(* PLC project passing_sensor, Dassault Systèmes ControlBuild 2024x *)
(* stored: creationDateTime 2023-10-03T11:13:57-01:00 *)

FUNCTION_BLOCK tri_chain.passing_sensor
  VAR_INPUT
    sensorSupply : BOOL := true;
  END_VAR
  VAR_OUTPUT
    passing : BOOL := false;
  END_VAR
  VAR
    status_act_prod : DINT := 0;
    m11 : REAL := 1.0;
    m12 : REAL := 0.0;
    m13 : REAL := 0.0;
    m14 : REAL := 0.0;
    m21 : REAL := 0.0;
    m22 : REAL := 1.0;
    m23 : REAL := 0.0;
    m24 : REAL := 0.0;
    m31 : REAL := 0.0;
    m32 : REAL := 0.0;
    m33 : REAL := 1.0;
    m34 : REAL := 0.0;
    m41 : REAL := 0.0;
    m42 : REAL := 0.0;
    m43 : REAL := 0.0;
    m44 : REAL := 1.0;
    px : REAL := 0.0;
    py : REAL := 0.0;
    pz : REAL := 0.0;
    dx : REAL := 0.0;
    dy : REAL := 0.0;
    dz : REAL := 0.0;
    detection : BOOL := false;
  END_VAR
  VAR CONSTANT
    passingLogic : BOOL := true;
  END_VAR
  VAR
    d_passing : BOOL := false;
    v_d_passing : BOOL := true;
  END_VAR


ACTION C_source_code:
/* ----------------------------------------------------------------	*/
/* Type : Model of Operative Behaviour					*/
/* Category :  Sensors							*/
/* Author : Dassault Systemes						*/
/* Update date : June 2018							*/
/* ----------------------------------------------------------------	*/
/* This module simulates the bahaviour of a  passing sensor 		*/
/*	for products.								*/
/* This module is an "actor".						*/
/* If it interacts with a product, this latter will acts on the	*/
/*	detection variable .							*/
/* -----------------------------------------------------------------	*/

/* -----------------------------------------------------------------	*/
/* "cptpass" module can be dragged in rotation or translation.	*/
/*	Then position and dimension variables can changed.		*/
/*	Then theses variables must be initialized from the data 	*/
/*	which are stored as parameters.					*/
/* -----------------------------------------------------------------	*/

if (d_passing) passing = v_d_passing;
else
	if ( sensorSupply ) passing=(detection ^ ! passingLogic);
	else passing = 0;

detection=0;
END_ACTION

ACTION C_header:

END_ACTION
END_FUNCTION_BLOCK
